Yaskawa INFORM job: SHIP2010.JBI

/JOB
//NAME SHIP2010
///FOLDERNAME MASTER
//POS
///NPOS 1,0,0,0,0,0
///TOOL 0
///POSTYPE PULSE
///PULSE
C00000=87036,-169218,-131221,87817,-127566,-310
//INST
///DATE 2021/10/29 11:49
///COMM YMCL MA1440 SHIPPING JOB V1.0
///ATTR SC,RO
///GROUP1 RB1
NOP
'*****************************
'USE THIS JOB TO POSITION THE
'ROBOT FOR INSTALLATION OF
'SHIPPING BRACKETS.
'*****************************
MOVJ C00000 VJ=5.00
END
